// SIMATIC S7-200 project (STEP 7-Micro/WIN), CPU 222 REL 01.22

SYMBOL_TABLE USR1
Always_On        SM0.0    // This bit is always on.
First_Scan_On    SM0.1    // This bit is on for the first scan cycle only.
P0_Config        SMB30    // Configure comm. port 0 (Freeport operation): baud rate, parity, # of data bits.
END_SYMBOL_TABLE

ORGANIZATION_BLOCK MAIN:OB1
TITLE=题目：S7-200与PC之间的连接：从WINDOWS应用程序中读数据
// ***概述***
// 这是一个用于小型泵站自动化控制的 PLC 程序，运行在 SIMATIC S7-200 CPU214 上，通过自由通信口与 Windows 应用程序（如 Microsoft Excel）通信，用于实时监控泵站运行状态。
// ***硬件和软件要求***
// 型号：SIMATIC CPU214或212                             
// ***软件***
// Software Wedge for Windows:
// Professional Edition Part #SW20WP或其他支持
// DDE Link的基于Windows的兼容软件
// ***程序注释***
// 设置通信口参数为 9600 波特、无奇偶校验、8 位字符。
// 绑定紧急阀开关的上升沿和下降沿到中断，并启用中断。
// 每当主泵开关上升沿时，发送 "Pump 1 is on"。
// 当主阀开关、主泵开关和紧急阀开关接通时，每秒增加计时器值，并更新其整数和十六进制表示。
// 发送缓冲区每秒更新，包含 "Flow time in sec:" 以及计时器的整数和十六进制值。
// 如果计时器超过 9999，复位计时器为 0。
// 若紧急阀开关上升沿触发，则发送 "Valve open"。
// 若紧急阀开关下降沿触发，则发送 "Valve closed"。
// 当紧急阀开关状态变化时，发送相应的阀状态信息。
BEGIN
Network 1 // ***主程序***
LD     First_Scan_On:SM0.1   // 首次扫描
CALL   SBR_0:SBR0            // 调用SBR0
Network 2
LD     I0.0                  //  若主泵开关I0.0=1
EU                           // 且上升沿
CALL   SBR_1:SBR1            // 则调用SBR1
Network 3
LD     I0.2                  // 若主阀开关I0.2=1
EU                           // 且上升沿
MOVW   +0, VW10              // 则定时器置0
Network 4
LD     I0.2                  // 若主阀开关I0.2=1
A      I0.0                  // 且泵运转(I0.0=1)
A      I0.1                  // 且紧急阀打开(I0.1=1)
CALL   SBR_2:SBR2            // 调用SBR2
Network 5 //  主程序结束
// 		
// 
END_ORGANIZATION_BLOCK

SUBROUTINE_BLOCK SBR_0:SBR0
TITLE=
BEGIN
Network 1 //  
LD     Always_On:SM0.0       // SM0.0总是1
MOVB   9, P0_Config:SMB30    // 自由通信口模式，9600波特，无奇偶校验
//每字符8位
ATCH   INT_0:INT0, 2         // 指定中断事件2(I0.1上升沿)调用中断程序0
ATCH   INT_1:INT1, 3         // 指定中断事件3(I0.1下降沿)调用中断程序1
ENI                          // 允许中断
Network 2 //  返回主程序
// RET				
// 
END_SUBROUTINE_BLOCK

SUBROUTINE_BLOCK SBR_1:SBR1
TITLE=
BEGIN
Network 1
LD     Always_On:SM0.0       // SM0.0总是1
MOVB   14, VB80              // 置发送信息长度（14个字节）
MOVD   16#50756D70, VD81     // 十六进制信息"Pump"
MOVD   16#20312069, VD85     // " 1 i"
MOVD   16#73206F6E, VD89     // "s on"
MOVW   16#D0A, VW93          // 回车换行表示信息结束
XMT    VB80, 0               // 发送(VB80中已存放所发送信息的字节数)
Network 2 //  返回主程序
// RET				
// 
END_SUBROUTINE_BLOCK

SUBROUTINE_BLOCK SBR_2:SBR2
TITLE=
BEGIN
Network 1
LD     Always_On:SM0.0       // SM0.0总为1
TON    T32, +1000            // 起动定时器T32(1000ms).
Network 2 //  
LD     T32                   // 一秒以后
MOVB   28, VB120             // 置发送信息长度(28个字节)
MOVD   16#466C6F77, VD121    // 
// "Flow"
MOVD   16#2074696D, VD125    // " tim"
MOVD   16#6520696E, VD129    // "e in"
MOVD   16#20736563, VD133    // " sec"
MOVB   16#3A, VB137          // ":" (字段分界符)
MOVB   16#3A, VB142          // ":" (字段分界符)
MOVW   16#D0A, VW147         // 回车换行表示信息结束
INCW   VW10                  // VW10增加1
MOVW   VW10, VW20            // 把VW10拷贝到VW20
IBCD   VW20                  // 把VW20转换成BCD码
HTA    VB20, VB138, 4        // 把BCD转换成ASCII(作数值显示)装入发送缓冲区
HTA    VB10, VB143, 4        // 把十六进制转换成ASCII(作十六进制显示)装入
//    发送缓冲区
XMT    VB120, 0              // 发送(VB120中已存放所发送信息的字节数)
MOVW   +0, T32               // 复位定时器
Network 3 //  
LDW=   VW10, +9999           // 若流出时间超出9999秒
MOVW   +0, VW10              // 则复位秒计数器
Network 4 //  返回主程序
// RET					
// 
END_SUBROUTINE_BLOCK

INTERRUPT_BLOCK INT_0:INT0
TITLE=
BEGIN
Network 1
LD     I0.0                  // 
MOVB   12, VB100             // 置发送信息长度（12个字节）
MOVD   16#56616C76, VD101    // 
// "Valv"
MOVD   16#653A6F70, VD105    // "e:op"
// ':' 是字段分界符
MOVD   16#656E0D0A, VD109    // "en"
// 回车换行表示信息结束
XMT    VB100, 0              // 发送(VB100中已存放所发送信息的字节数)
Network 2 //  返回主程序
// RET					
// 
END_INTERRUPT_BLOCK

INTERRUPT_BLOCK INT_1:INT1
TITLE=
BEGIN
Network 2
LD     I0.0                  // SM0.0总位1
MOVB   14, VB100             // 置发送信息长度(14个字节)
MOVD   16#56616C76, VD101    // 
// "Valv"
MOVD   16#653A636C, VD105    // "e cl"
MOVD   16#6F736564, VD109    // "osed"
MOVW   16#D0A, VW113         // 回车换行表示信息结束
XMT    VB100, 0              // 发送(VB100中已存放所发送信息的字节数)
Network 3 //  返回主程序
// RET					
// 
END_INTERRUPT_BLOCK
